{attribute 'GeneratedUsingTerminal: KL3152'}
{attribute addProperty BoxType "KL3152"}
{attribute addProperty Description ""}
{attribute addProperty Physics ""}
{attribute addProperty Id "Channel_1AT %Q*Channel_03CEAA5E0Channel_2AT %Q*Channel_03CEAA5E0"}
{attribute addProperty CRC "2016972219"}
{attribute addProperty Size "0"}
TYPE KL3152_78388DBB :
STRUCT
	{attribute addProperty Name "Channel_1"}
	Channel_1 : Channel_03CEAA5E;
	{attribute addProperty Name "Channel_2"}
	Channel_2 : Channel_03CEAA5E;
END_STRUCT
END_TYPE

(* stored: Version 1.2.0.0, ProductVersion 3.1.4024.9
   DUT KL3152_78388DBB: Id {70a69195-842c-4582-ad37-62d56bba1896} *)
